PROGRAM MAIN
VAR
	LidApplicatiorCylinder : T_Cylinder;
	LidApplyStation : T_LidApplyStation(Cylinder := LidApplicatiorCylinder);

	start: BOOL;
END_VAR

LidApplyStation();

IF start THEN
	start := FALSE;
	LidApplyStation.Start();
END_IF

END_PROGRAM

(* stored: Version 1.1.0.1, ProductVersion 3.1.4024.4
   POU MAIN: Id {1e6b7d9a-faea-47b8-b7fd-cf99fa7903a5}, SpecialFunc None *)
